// TIA Portal V18 export
ORGANIZATION_BLOCK "18-Cab Floor"   // OB127, LAD, ProgramCycle
TITLE = "Main Program Sweep (Cycle)"
{ S7_Optimized_Access := 'TRUE' }
VERSION : 0.1
// stored: AutoNumber true, IsIECCheckEnabled false, SetENOAutomatically false
   VAR_INPUT
      Initial_Call : Bool;   // Initial call of this OB
      Remanence : Bool;   // =True, if remanent data are available
   END_VAR
   VAR_TEMP   // added for the SCL form of the ladder/FBD networks
      _w1 : Bool;
   END_VAR
BEGIN

REGION Network 1: Cab Floor Control Manuel & Auto
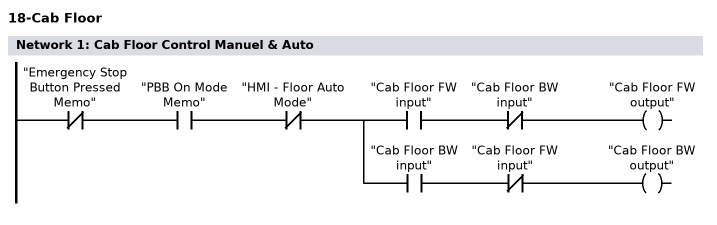
   RUNG wire#powerrail
      I_Contact( "Emergency Stop Button Pressed Memo" )
      Contact( "PBB On Mode Memo" )
      I_Contact( "HMI - Floor Auto Mode" )
      wire#w1
      Contact( "Cab Floor FW input" )
      I_Contact( "Cab Floor BW input" )
      Coil( "Cab Floor FW output" )
   END_RUNG
   RUNG wire#w1
      Contact( "Cab Floor BW input" )
      I_Contact( "Cab Floor FW input" )
      Coil( "Cab Floor BW output" )
   END_RUNG
   // the same network as SCL:
   #_w1 := NOT "Emergency Stop Button Pressed Memo" AND "PBB On Mode Memo" AND NOT "HMI - Floor Auto Mode";
   "Cab Floor FW output" := #_w1 AND "Cab Floor FW input" AND NOT "Cab Floor BW input";
   "Cab Floor BW output" := #_w1 AND "Cab Floor BW input" AND NOT "Cab Floor FW input";
END_REGION
END_ORGANIZATION_BLOCK
